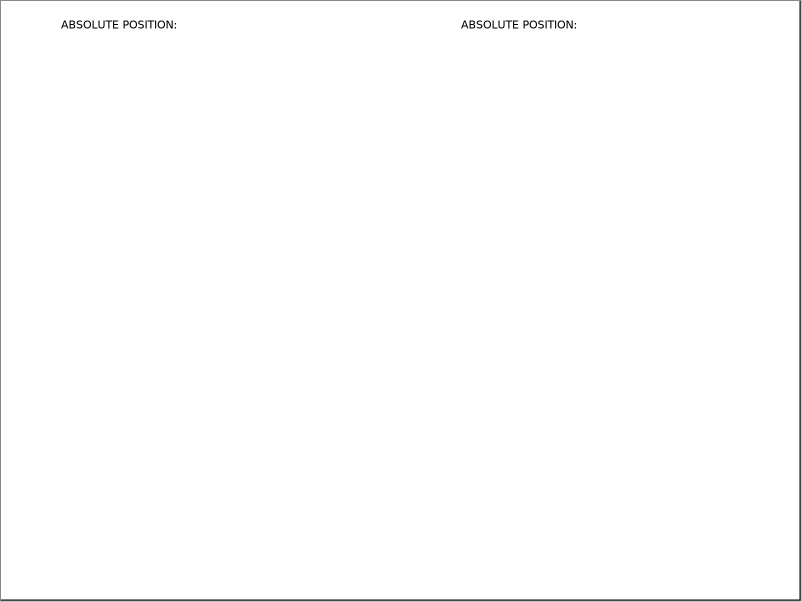
VISUALIZATION F38_Velocity_Profile  // 802x602
    Rectangle (0,0 800x600)
    Label (10,10 170x30), "ABSOLUTE POSITION:"
    Label (410,10 170x30), "ABSOLUTE POSITION:"
END_VISUALIZATION

(* stored: Version 1.1.0.1, ProductVersion 3.1.4022.7
   Visu F38_Velocity_Profile: Id {32a9dabe-64fe-40b7-aaf1-57faf63e1127} *)
